// TIA Portal V16 export
// export: Created 2024-08-29T13:25:47.1543466Z, ExportSetting WithDefaults, DisplayName Totally Integrated Automation Portal, DisplayVersion V16, DisplayName TIA Portal Version Control Interface, DisplayVersion V16, DisplayName TIA Portal Openness, DisplayVersion V16, DisplayName STEP 7 Professional, DisplayVersion V16, DisplayName STEP 7 Safety, DisplayVersion V16, DisplayName WinCC Professional, DisplayVersion V16
TYPE "UT00802_St_ConstAqRawData"
TITLE = Static UDT [SYSTEM CONSTANTS] — Analog Input Card Types, Ranges and Coefficients
// PRACTICAL SERIES AUTOMATION LIBRARY (PAL)   —   COPYRIGHT 2020 – M. GLEDHILL (MIT LICENCE)
//                   ———— ◆ ————
// FULL ONLINE DOCUMENTATION IS AVAILABLE AT: https://practicalseries.com/2001-pal/index.html
// stored: IsFailsafeCompliant false
   STRUCT
      revInfo { ExternalWritable := 'False'} : "UT01000_St_SysRevision";   // ▀▀▀▀ UDT CURRENT REVISION
      ___________0010_0 { ExternalAccessible := 'False'; ExternalVisible := 'False'; ExternalWritable := 'False'} : Bool;
      ___________0010_1 { ExternalAccessible := 'False'; ExternalVisible := 'False'; ExternalWritable := 'False'} : Bool;   // ▀▀▀▀ AQ SIGNAL CODE
      AQ_CODE { ExternalWritable := 'False'} : UInt := 16#0000;   // Input code (type, coefficient and range)
      ___________0020_0 { ExternalAccessible := 'False'; ExternalVisible := 'False'; ExternalWritable := 'False'} : Bool := false;
      ___________0020_1 { ExternalAccessible := 'False'; ExternalVisible := 'False'; ExternalWritable := 'False'} : Bool;   // ▀▀▀▀ AQ RANGE DATA
      RAW_MIN { ExternalWritable := 'False'} : Int := 0;   // Minimum value of the analog input range
      RAW_MAX { ExternalWritable := 'False'} : Int := 27648;   // Maximum value of the analog input range
      RAW_DESC { ExternalWritable := 'False'} : String[60] := 'User defined instrument type';   // Signal type description (plain English)
      ___________0030_1 { ExternalAccessible := 'False'; ExternalVisible := 'False'; ExternalWritable := 'False'} : Bool;
      ___________0030_2 { ExternalAccessible := 'False'; ExternalVisible := 'False'; ExternalWritable := 'False'} : Bool;   // ▀▀▀▀ AQ CARD PARAMETERS
      PARAM_TYPE { ExternalWritable := 'False'} : Byte := 16#00;   // Unique measurement type code
      PARAM_RANGE { ExternalWritable := 'False'} : Byte := 16#00;   // Unique measurement range code
   END_STRUCT;
   // revInfo.REV_BLOCK := 'UT00802';
   // revInfo.REV_NUMBER := '001.000';
   // revInfo.REV_DATE := '2024-05-16';
   // revInfo.REV_AUTHOR := 'M. Gledhill';
END_TYPE
